# B&R Automation Studio project EFI (part 2)

### IoMap.iom - X20CP1382/IoMap.iom
```iecst
VAR_CONFIG
	Cyclic#4.::X20DIF371_002.DInput[1] AT %IX."X20DIF371_002".DigitalInput01;
	Cyclic#4.::X20DIF371_002.DInput[2] AT %IX."X20DIF371_002".DigitalInput02;
	Cyclic#4.::X20DIF371_002.DInput[3] AT %IX."X20DIF371_002".DigitalInput03;
	Cyclic#4.::X20DIF371_002.DInput[4] AT %IX."X20DIF371_002".DigitalInput04;
	Cyclic#4.::X20DIF371_002.DInput[5] AT %IX."X20DIF371_002".DigitalInput05;
	Cyclic#4.::X20DIF371_002.DInput[6] AT %IX."X20DIF371_002".DigitalInput06;
	Cyclic#4.::X20DIF371_002.DInput[7] AT %IX."X20DIF371_002".DigitalInput07;
	Cyclic#4.::X20DIF371_002.DInput[8] AT %IX."X20DIF371_002".DigitalInput08;
	Cyclic#4.::X20DIF371_002.DInput[9] AT %IX."X20DIF371_002".DigitalInput09;
	Cyclic#4.::X20DIF371_002.DInput[10] AT %IX."X20DIF371_002".DigitalInput10;
	Cyclic#4.::X20DIF371_002.DInput[11] AT %IX."X20DIF371_002".DigitalInput11;
	Cyclic#4.::X20DIF371_002.DInput[12] AT %IX."X20DIF371_002".DigitalInput12;
	Cyclic#4.::X20DIF371_002.DInput[13] AT %IX."X20DIF371_002".DigitalInput13;
	Cyclic#4.::X20DIF371_002.DInput[14] AT %IX."X20DIF371_002".DigitalInput14;
	Cyclic#4.::X20DIF371_002.DInput[15] AT %IX."X20DIF371_002".DigitalInput15;
	Cyclic#4.::X20DIF371_002.DInput[16] AT %IX."X20DIF371_002".DigitalInput16;
	Cyclic#4.::X20DIF371_001.ModuleOk AT %IX."X20DIF371_001".ModuleOk;
	Cyclic#2.::X1.DInput[1] AT %IX."X1".DigitalInput01;
	Cyclic#2.::X1.DInput[2] AT %IX."X1".DigitalInput02;
	Cyclic#2.::X1.DInput[3] AT %IX."X1".DigitalInput03;
	Cyclic#4.::X1.DInput[4] AT %IX."X1".DigitalInput04;
	Cyclic#4.::X1.AInput[1] AT %IW."X1".AnalogInput01;
	Cyclic#4.::X1.AInput[2] AT %IW."X1".AnalogInput02;
	Cyclic#4.::X1.Status01 AT %IB."X1".StatusInput01;
	Cyclic#4.::X2.DInput[1] AT %IX."X2".DigitalInput01;
	Cyclic#4.::X2.DInput[2] AT %IX."X2".DigitalInput02;
	Cyclic#4.::X2.DInput[3] AT %IX."X2".DigitalInput03;
	Cyclic#4.::X2.DInput[4] AT %IX."X2".DigitalInput04;
	Cyclic#4.::X2.DInput[5] AT %IX."X2".DigitalInput05;
	Cyclic#4.::X2.DInput[6] AT %IX."X2".DigitalInput06;
	Cyclic#4.::X2.DInput[7] AT %IX."X2".DigitalInput07;
	Cyclic#4.::X2.DInput[8] AT %IX."X2".DigitalInput08;
	Cyclic#4.::X2.DInput[9] AT %IX."X2".DigitalInput09;
	Cyclic#4.::X2.DInput[10] AT %IX."X2".DigitalInput10;
	Cyclic#4.::X2.DInput[11] AT %IX."X2".DigitalInput11;
	Cyclic#4.::X2.DInput[12] AT %IX."X2".DigitalInput12;
	Cyclic#4.::X2.DInput[13] AT %IX."X2".DigitalInput13;
	Cyclic#4.::X2.DInput[14] AT %IX."X2".DigitalInput14;
	Cyclic#4.::X20DIF371_002.ModuleOk AT %IX."X20DIF371_002".ModuleOk;
	Cyclic#4.::X20DIF371_003.DInput[1] AT %IX."X20DIF371_003".DigitalInput01;
	Cyclic#4.::X20DIF371_003.DInput[2] AT %IX."X20DIF371_003".DigitalInput02;
	Cyclic#4.::X20DIF371_003.DInput[3] AT %IX."X20DIF371_003".DigitalInput03;
	Cyclic#4.::X20DIF371_003.DInput[4] AT %IX."X20DIF371_003".DigitalInput04;
	Cyclic#4.::X20DIF371_003.DInput[5] AT %IX."X20DIF371_003".DigitalInput05;
	Cyclic#4.::X20DIF371_003.DInput[6] AT %IX."X20DIF371_003".DigitalInput06;
	Cyclic#4.::X20DIF371_003.DInput[7] AT %IX."X20DIF371_003".DigitalInput07;
	Cyclic#4.::X20DIF371_003.DInput[8] AT %IX."X20DIF371_003".DigitalInput08;
	Cyclic#4.::X20DIF371_003.DInput[9] AT %IX."X20DIF371_003".DigitalInput09;
	Cyclic#4.::X20DIF371_003.DInput[10] AT %IX."X20DIF371_003".DigitalInput10;
	Cyclic#4.::X20DIF371_003.DInput[11] AT %IX."X20DIF371_003".DigitalInput11;
	Cyclic#4.::X20DIF371_003.DInput[12] AT %IX."X20DIF371_003".DigitalInput12;
	Cyclic#4.::X20DIF371_003.DInput[13] AT %IX."X20DIF371_003".DigitalInput13;
	Cyclic#4.::X20DIF371_003.DInput[14] AT %IX."X20DIF371_003".DigitalInput14;
	Cyclic#4.::X20DIF371_003.DInput[15] AT %IX."X20DIF371_003".DigitalInput15;
	Cyclic#4.::X20DIF371_003.DInput[16] AT %IX."X20DIF371_003".DigitalInput16;
	Cyclic#4.::X20DIF371_004.ModuleOk AT %IX."X20DIF371_004".ModuleOk;
	Cyclic#1.::SiUnitBK1.ModuleOk AT %IX."SI_unit_BK1".ModuleOk;
	Cyclic#1.::SiUnitBK1.NodeStatus AT %IW."SI_unit_BK1".NodeStatus;
	Cyclic#1.::SiUnitBK1.Input01_08 AT %IB."SI_unit_BK1".ReadInout1hTo8h_6000sub1;
	Cyclic#1.::SiUnitBK1.Input09_16 AT %IB."SI_unit_BK1".ReadInput9hTo16h_6000sub2;
	Cyclic#1.::SiUnitBK1.Input17_24 AT %IB."SI_unit_BK1".ReadInput17hTo24h_6000sub3;
	Cyclic#1.::SiUnitBK1.Input25_32 AT %IB."SI_unit_BK1".ReadInput25hTo32h_6000sub4;
	Cyclic#1.::SiUnitBK1.Output01_08 AT %QB."SI_unit_BK1".WriteOutput1hTo8h_6200sub1;
	Cyclic#1.::SiUnitBK1.Output09_16 AT %QB."SI_unit_BK1".WriteOutput9hTo16h_6200sub2;
	Cyclic#1.::SiUnitBK1.Output17_24 AT %QB."SI_unit_BK1".WriteOutput17hTo24h_6200sub3;
	Cyclic#1.::SiUnitBK1.Output25_32 AT %QB."SI_unit_BK1".WriteOutput25hTo32h_6200sub4;
	Cyclic#4.::X3.DInput[5] AT %IX."X3".DigitalInput05;
	Cyclic#4.::X3.DInput[6] AT %IX."X3".DigitalInput06;
	Cyclic#4.::X3.DInput[7] AT %IX."X3".DigitalInput07;
	Cyclic#4.::X3.DOutput[1] AT %QX."X3".DigitalOutput01;
	Cyclic#4.::X3.DOutput[2] AT %QX."X3".DigitalOutput02;
	Cyclic#4.::X3.DOutput[3] AT %QX."X3".DigitalOutput03;
	Cyclic#4.::X3.DOutput[4] AT %QX."X3".DigitalOutput04;
	Cyclic#4.::X3.DOutput[8] AT %QX."X3".DigitalOutput08;
	Cyclic#4.::X3.DOutput[9] AT %QX."X3".DigitalOutput09;
	Cyclic#4.::X3.DOutput[10] AT %QX."X3".DigitalOutput10;
	Cyclic#4.::X3.DOutput[11] AT %QX."X3".DigitalOutput11;
	Cyclic#4.::X3.DOutput[12] AT %QX."X3".DigitalOutput12;
	Cyclic#4.::X20DOF322_005.ModuleOk AT %IX."X20DOF322_005".ModuleOk;
	Cyclic#1.::gIclaNetData[1].xModuleOK AT %IX."ILE1F_BK1".ModuleOk;
	Cyclic#1.::gIclaNetData[1].RPDO4.driveCtrl AT %QB."ILE1F_BK1".Pdo4_driveCtrl_301Esub1;
	Cyclic#1.::gIclaNetData[1].RPDO4.modeCtrl AT %QB."ILE1F_BK1".Pdo4_modeCtrl_301Esub2;
	Cyclic#1.::gIclaNetData[1].TPDO4.modeStat AT %IB."ILE1F_BK1".Pdo4_modeStat_301Esub3;
	Cyclic#1.::gIclaNetData[1].TPDO4.driveStat AT %IW."ILE1F_BK1".Pdo4_driveStat_301Esub4;
	Cyclic#1.::gIclaNetData[1].RPDO4.Ref16 AT %QW."ILE1F_BK1".Pdo4_Ref16_301Esub5;
	Cyclic#1.::gIclaNetData[1].RPDO4.Ref32 AT %QD."ILE1F_BK1".Pdo4_Ref32_301Esub6;
	Cyclic#1.::gIclaNetData[1].TPDO4.Act32 AT %ID."ILE1F_BK1".Pdo4_Act32_301Esub8;
	Cyclic#1.::gIclaNetData[1].TPDO4.Act8 AT %IB."ILE1F_BK1".Pdo4_Act8_301Esub7;
	Cyclic#1.::gAxisStepper[1].DrvIf.iLifeCnt AT %IB."X20SM1436_011".LifeCnt;
	Cyclic#1.::gAxisStepper[1].DrvIf.iDrvOK AT %IX."X20SM1436_011".DrvOk01;
	Cyclic#1.::gAxisStepper[1].DrvIf.oBoostCurrent AT %QX."X20SM1436_011".BoostCurrent01;
	Cyclic#1.::gAxisStepper[1].DrvIf.oStandStillCurrent AT %QX."X20SM1436_011".StandstillCurrent01;
	Cyclic#1.::gAxisStepper[1].DrvIf.oSetTime AT %QW."X20SM1436_011".SetTime01;
	Cyclic#1.::gAxisStepper[1].DiDoIf.iLifeCntDriveEnable AT %IB."X20SM1436_011".LifeCnt;
	Cyclic#1.::gAxisStepper[1].DiDoIf.iLifeCntDriveReady AT %IB."X20SM1436_011".LifeCnt;
	Cyclic#1.::gAxisStepper[1].DiDoIf.iDriveReady AT %IX."X20SM1436_011".DrvOk01;
	Cyclic#1.::gAxisStepper[1].EncIf1.iLifeCnt AT %IB."X20SM1436_011".LifeCnt;
	Cyclic#1.::gAxisStepper[1].EncIf1.iEncOK AT %IX."X20SM1436_011".EncOk01;
	Cyclic#1.::gAxisStepper[1].EncIf1.iActPos AT %IW."X20SM1436_011".ActPos01;
	Cyclic#1.::gAxisStepper[1].EncIf1.iRefPulsePos AT %IW."X20SM1436_011".RefPulsePos01;
	Cyclic#1.::gAxisStepper[1].EncIf1.iRefPulseCnt AT %IB."X20SM1436_011".RefPulseCnt01;
	Cyclic#1.::gAxisStepper[1].EncIf1.iActTime AT %IW."X20SM1436_011".ActTime01;
	Cyclic#1.::X20SM1436_011.ModuleOk AT %IX."X20SM1436_011".ModuleOk;
	Cyclic#1.::gAxisStepper[1].DiDoIf.oDriveEnable AT %QX."X20SM1436_011".DriveEnable01;
	Cyclic#1.::gAxisStepper[1].MotorStep0 AT %QW."X20SM1436_011".Motor1Step0;
	Cyclic#1.::gAxisStepper[2].DrvIf.iLifeCnt AT %IB."X20SM1436_012".LifeCnt;
	Cyclic#1.::gAxisStepper[2].DrvIf.iDrvOK AT %IX."X20SM1436_012".DrvOk01;
	Cyclic#1.::gAxisStepper[2].DrvIf.oBoostCurrent AT %QX."X20SM1436_012".BoostCurrent01;
	Cyclic#1.::gAxisStepper[2].DrvIf.oStandStillCurrent AT %QX."X20SM1436_012".StandstillCurrent01;
	Cyclic#1.::gAxisStepper[2].DrvIf.oSetTime AT %QW."X20SM1436_012".SetTime01;
	Cyclic#1.::gAxisStepper[2].MotorStep0 AT %QW."X20SM1436_012".Motor1Step0;
	Cyclic#1.::gAxisStepper[2].DiDoIf.iLifeCntDriveEnable AT %IB."X20SM1436_012".LifeCnt;
	Cyclic#1.::gAxisStepper[2].DiDoIf.iLifeCntDriveReady AT %IB."X20SM1436_012".LifeCnt;
	Cyclic#1.::gAxisStepper[2].DiDoIf.iDriveReady AT %IX."X20SM1436_012".DrvOk01;
	Cyclic#1.::gAxisStepper[2].DiDoIf.oDriveEnable AT %QX."X20SM1436_012".DriveEnable01;
	Cyclic#1.::gAxisStepper[2].EncIf1.iLifeCnt AT %IB."X20SM1436_012".LifeCnt;
	Cyclic#1.::gAxisStepper[2].EncIf1.iEncOK AT %IX."X20SM1436_012".EncOk01;
	Cyclic#1.::gAxisStepper[2].EncIf1.iActPos AT %IW."X20SM1436_012".ActPos01;
	Cyclic#1.::gAxisStepper[2].EncIf1.iRefPulsePos AT %IW."X20SM1436_012".RefPulsePos01;
	Cyclic#1.::gAxisStepper[2].EncIf1.iRefPulseCnt AT %IB."X20SM1436_012".RefPulseCnt01;
	Cyclic#1.::gAxisStepper[2].EncIf1.iActTime AT %IW."X20SM1436_012".ActTime01;
	Cyclic#1.::X20SM1436_012.ModuleOk AT %IX."X20SM1436_012".ModuleOk;
	Cyclic#4.::X20DIF371_001.DInput[1] AT %IX."X20DIF371_001".DigitalInput01;
	Cyclic#4.::X20DIF371_001.DInput[2] AT %IX."X20DIF371_001".DigitalInput02;
	Cyclic#4.::X20DIF371_001.DInput[3] AT %IX."X20DIF371_001".DigitalInput03;
	Cyclic#4.::X20DIF371_001.DInput[4] AT %IX."X20DIF371_001".DigitalInput04;
	Cyclic#4.::X20DIF371_001.DInput[5] AT %IX."X20DIF371_001".DigitalInput05;
	Cyclic#4.::X20DIF371_001.DInput[6] AT %IX."X20DIF371_001".DigitalInput06;
	Cyclic#4.::X20DIF371_001.DInput[7] AT %IX."X20DIF371_001".DigitalInput07;
	Cyclic#4.::X20DIF371_001.DInput[8] AT %IX."X20DIF371_001".DigitalInput08;
	Cyclic#4.::X20DIF371_001.DInput[9] AT %IX."X20DIF371_001".DigitalInput09;
	Cyclic#4.::X20DIF371_001.DInput[10] AT %IX."X20DIF371_001".DigitalInput10;
	Cyclic#4.::X20DIF371_001.DInput[11] AT %IX."X20DIF371_001".DigitalInput11;
	Cyclic#4.::X20DIF371_001.DInput[12] AT %IX."X20DIF371_001".DigitalInput12;
	Cyclic#4.::X20DIF371_001.DInput[13] AT %IX."X20DIF371_001".DigitalInput13;
	Cyclic#4.::X20DIF371_001.DInput[14] AT %IX."X20DIF371_001".DigitalInput14;
	Cyclic#4.::X20DIF371_001.DInput[15] AT %IX."X20DIF371_001".DigitalInput15;
	Cyclic#4.::X20DIF371_001.DInput[16] AT %IX."X20DIF371_001".DigitalInput16;
	::X20DIF371_003.ModuleOk AT %IX."X20DIF371_003".ModuleOk;
	Cyclic#4.::X20DIF371_004.DInput[1] AT %IX."X20DIF371_004".DigitalInput01;
	Cyclic#4.::X20DIF371_004.DInput[2] AT %IX."X20DIF371_004".DigitalInput02;
	Cyclic#4.::X20DIF371_004.DInput[3] AT %IX."X20DIF371_004".DigitalInput03;
	Cyclic#4.::X20DIF371_004.DInput[4] AT %IX."X20DIF371_004".DigitalInput04;
	Cyclic#4.::X20DIF371_004.DInput[5] AT %IX."X20DIF371_004".DigitalInput05;
	Cyclic#4.::X20DIF371_004.DInput[6] AT %IX."X20DIF371_004".DigitalInput06;
	Cyclic#4.::X20DIF371_004.DInput[7] AT %IX."X20DIF371_004".DigitalInput07;
	Cyclic#4.::X20DIF371_004.DInput[8] AT %IX."X20DIF371_004".DigitalInput08;
	Cyclic#4.::X20DIF371_004.DInput[9] AT %IX."X20DIF371_004".DigitalInput09;
	Cyclic#4.::X20DIF371_004.DInput[10] AT %IX."X20DIF371_004".DigitalInput10;
	Cyclic#4.::X20DIF371_004.DInput[11] AT %IX."X20DIF371_004".DigitalInput11;
	Cyclic#4.::X20DIF371_004.DInput[12] AT %IX."X20DIF371_004".DigitalInput12;
	Cyclic#4.::X20DIF371_004.DInput[13] AT %IX."X20DIF371_004".DigitalInput13;
	Cyclic#4.::X20DIF371_004.DInput[14] AT %IX."X20DIF371_004".DigitalInput14;
	Cyclic#4.::X20DIF371_004.DInput[15] AT %IX."X20DIF371_004".DigitalInput15;
	Cyclic#4.::X20DIF371_004.DInput[16] AT %IX."X20DIF371_004".DigitalInput16;
	Cyclic#4.::X20DOF322_005.DOutput[1] AT %QX."X20DOF322_005".DigitalOutput01;
	Cyclic#4.::X20DOF322_005.DOutput[2] AT %QX."X20DOF322_005".DigitalOutput02;
	Cyclic#4.::X20DOF322_005.DOutput[3] AT %QX."X20DOF322_005".DigitalOutput03;
	Cyclic#4.::X20DOF322_005.DOutput[4] AT %QX."X20DOF322_005".DigitalOutput04;
	Cyclic#4.::X20DOF322_005.DOutput[5] AT %QX."X20DOF322_005".DigitalOutput05;
	Cyclic#4.::X20DOF322_005.DOutput[6] AT %QX."X20DOF322_005".DigitalOutput06;
	Cyclic#4.::X20DOF322_005.DOutput[7] AT %QX."X20DOF322_005".DigitalOutput07;
	Cyclic#4.::X20DOF322_005.DOutput[8] AT %QX."X20DOF322_005".DigitalOutput08;
	Cyclic#4.::X20DOF322_005.DOutput[9] AT %QX."X20DOF322_005".DigitalOutput09;
	Cyclic#4.::X20DOF322_005.DOutput[10] AT %QX."X20DOF322_005".DigitalOutput10;
	Cyclic#4.::X20DOF322_005.DOutput[11] AT %QX."X20DOF322_005".DigitalOutput11;
	Cyclic#4.::X20DOF322_005.DOutput[12] AT %QX."X20DOF322_005".DigitalOutput12;
	Cyclic#4.::X20DOF322_005.DOutput[13] AT %QX."X20DOF322_005".DigitalOutput13;
	Cyclic#4.::X20DOF322_005.DOutput[14] AT %QX."X20DOF322_005".DigitalOutput14;
	Cyclic#4.::X20DOF322_005.DOutput[15] AT %QX."X20DOF322_005".DigitalOutput15;
	Cyclic#4.::X20DOF322_005.DOutput[16] AT %QX."X20DOF322_005".DigitalOutput16;
	::X20DOF322_006.ModuleOk AT %IX."X20DOF322_006".ModuleOk;
	Cyclic#4.::X20DOF322_006.DOutput[1] AT %QX."X20DOF322_006".DigitalOutput01;
	Cyclic#4.::X20DOF322_006.DOutput[2] AT %QX."X20DOF322_006".DigitalOutput02;
	Cyclic#4.::X20DOF322_006.DOutput[3] AT %QX."X20DOF322_006".DigitalOutput03;
	Cyclic#4.::X20DOF322_006.DOutput[4] AT %QX."X20DOF322_006".DigitalOutput04;
	Cyclic#4.::X20DOF322_006.DOutput[5] AT %QX."X20DOF322_006".DigitalOutput05;
	Cyclic#4.::X20DOF322_006.DOutput[6] AT %QX."X20DOF322_006".DigitalOutput06;
	Cyclic#4.::X20DOF322_006.DOutput[7] AT %QX."X20DOF322_006".DigitalOutput07;
	Cyclic#4.::X20DOF322_006.DOutput[8] AT %QX."X20DOF322_006".DigitalOutput08;
	Cyclic#4.::X20DOF322_006.DOutput[9] AT %QX."X20DOF322_006".DigitalOutput09;
	Cyclic#4.::X20DOF322_006.DOutput[10] AT %QX."X20DOF322_006".DigitalOutput10;
	Cyclic#4.::X20DOF322_006.DOutput[11] AT %QX."X20DOF322_006".DigitalOutput11;
	Cyclic#4.::X20DOF322_006.DOutput[12] AT %QX."X20DOF322_006".DigitalOutput12;
	Cyclic#4.::X20DOF322_006.DOutput[13] AT %QX."X20DOF322_006".DigitalOutput13;
	Cyclic#4.::X20DOF322_006.DOutput[14] AT %QX."X20DOF322_006".DigitalOutput14;
	Cyclic#4.::X20DOF322_006.DOutput[15] AT %QX."X20DOF322_006".DigitalOutput15;
	Cyclic#4.::X20DOF322_006.DOutput[16] AT %QX."X20DOF322_006".DigitalOutput16;
	Cyclic#4.::X20AO4622_009.ModuleOk AT %IX."X20AO4622_009".ModuleOk;
	Cyclic#4.::X20AO4622_009.AOutput[1] AT %QW."X20AO4622_009".AnalogOutput01;
	Cyclic#4.::X20AO4622_009.AOutput[2] AT %QW."X20AO4622_009".AnalogOutput02;
	Cyclic#4.::X20AO4622_009.AOutput[3] AT %QW."X20AO4622_009".AnalogOutput03;
	Cyclic#4.::X20AO4622_009.AOutput[4] AT %QW."X20AO4622_009".AnalogOutput04;
	Cyclic#4.::X20AT4222_010.ModuleOk AT %IX."X20AT4222_010".ModuleOk;
	Cyclic#4.::X20AT4222_010.TempInput[1] AT %IW."X20AT4222_010".Temperature01;
	Cyclic#4.::X20AT4222_010.TempInput[2] AT %IW."X20AT4222_010".Temperature02;
	Cyclic#4.::X20AT4222_010.TempInput[3] AT %IW."X20AT4222_010".Temperature03;
	Cyclic#4.::X20AT4222_010.TempInput[4] AT %IW."X20AT4222_010".Temperature04;
	X20AI4322_008.AInput[1] AT %IW."X20AI4322_008".AnalogInput01;
	X20AI4322_008.AInput[2] AT %IW."X20AI4322_008".AnalogInput02;
	X20AI4322_008.AInput[3] AT %IW."X20AI4322_008".AnalogInput03;
	X20AI4322_008.AInput[4] AT %IW."X20AI4322_008".AnalogInput04;
	X20AI4322_008.ModuleOk AT %IX."X20AI4322_008".ModuleOk;
	X20AI4322_008.Status01 AT %IB."X20AI4322_008".StatusInput01;
	::X20AT4222_010.Status01 AT %IB."X20AT4222_010".StatusInput01;
END_VAR
```

### Acp10cfg.ncc - X20CP1382/Motion/Acp10cfg.ncc
```
NcConfiguration (Version=5.15.1, NcSwId=Acp10)
  ACP10CF1_typ:
    cnt_nettrc_rec_drive = 1500
    bufsize_trace_upload = 1200
    tc_nc_man_task = Cyclic #1
    glob_pv_as_ncobject = Yes
    ncsys_dl_broadcast = Yes
    ncsys_dl_acp_reset = Yes
    safemc_log_err_to_ax = Yes
    network_init:
      ncsw_init_execute = Yes
      automatic_execute = Yes
      node_nr_warning = Yes
      net_err_before_ncact = Yes
    nettrc:
      enter_parsecrec = Yes
      enter_ncaction = Yes
      save_ring_startidx = No
    cam_prof_download:
      cam_dat_dl_parallel = No
      tc_cam_dl_parallel = Task class for NC Manager task
    plk_if[0]:
      if_name = IF3
      tc_CycDat_PLCopen = Task class for NC Manager task
      mc_broadcast_extdat = No
    sdc_if[0]:
      if_name = SDC_IF1
      mc_broadcast_size = 800
      mc_broadcast_extdat = No
```

### Acp10map.ncm - X20CP1382/Motion/Acp10map.ncm
```
NcMapping (NcSwId=Acp10, DisabledNodesAreHidden=False)
  NcObject gAxis01 (ModuleId=8V1045.00-2_BELT, Type=ncAXIS, Channel=1, AcoposSimulation=Off, InitParameter=BeltShiel1, AcoposParameter=BeltShield, Disabled=FALSE, ModuleDisabled=FALSE)
  NcObject 8V1045.00-2_ncV_AXIS1 (ModuleId=8V1045.00-2_BELT, Type=ncV_AXIS, Channel=1, Disabled=TRUE, ModuleDisabled=FALSE)
  NcObject gAxis21 (ModuleId=8V1010.50-2_BK1, Type=ncAXIS, Channel=1, AcoposSimulation=Off, InitParameter=BK1_i, AcoposParameter=BK1_a, Disabled=FALSE, ModuleDisabled=FALSE)
  NcObject 8V1016.50-2_ncV_AXIS1 (ModuleId=8V1010.50-2_BK1, Type=ncV_AXIS, Channel=1, Disabled=TRUE, ModuleDisabled=FALSE)
  NcObject gAxisStp01 (ModuleId=X20SM1436_011, ModuleAddress=SDC_IF1.ST1, Type=ncAXIS, Channel=1, AcoposSimulation=Off, InitParameter=SM_i, AcoposParameter=SM_a, AdditionalData=SDC_AX_HwPv="gAxisStepper[1].HW", Disabled=FALSE, ModuleDisabled=FALSE)
  NcObject gAxisStp02 (ModuleId=X20SM1436_012, ModuleAddress=SDC_IF1.ST2, Type=ncAXIS, Channel=1, AcoposSimulation=Off, InitParameter=SM_i, AcoposParameter=SM_a, AdditionalData=SDC_AX_HwPv="gAxisStepper[2].HW", Disabled=FALSE, ModuleDisabled=FALSE)
```

## Configuration 2BK12Bar

CPU X20CP1382, AutomationRuntime B4.83, Build 4.1.2, Safety 1.10, Vc V4.72.6

### Task classes (Cpu.sw)
```
Cyclic#1 (cycle 4000 us, tolerance 0 us):
  InitSteprs <- ExtPack._Motion.StepperCtrl.StepperCtrl_v1.InitStepperX2XCtrl.prg (BuildOptions=-D _IGNORE_CHECKLIB)
  Stepper3L1 <- ExtPack._Motion.StepperCtrl.StepperCtrl_v1.StepperX2XCtrl.prg (BuildOptions=-D _IGNORE_CHECKLIB)
  Stepper3L2 <- ExtPack._Motion.StepperCtrl.StepperCtrl_v1.StepperX2XCtrl.prg (BuildOptions=-D _IGNORE_CHECKLIB)
  Analog <- (binary) (BuildOptions=-D _IGNORE_CHECKLIB)
Cyclic#2 (cycle 12000 us, tolerance 0 us):
  Initialize <- Printer.Config.Initialize.prg (BuildOptions=-D _IGNORE_CHECKLIB)
  InitAxis <- ExtPack._Motion.AxisCtrl.AxisCtrl_v2.InitAxisControl.prg (BuildOptions=-D _IGNORE_CHECKLIB)
  Belt <- ExtPack._Motion.AxisCtrl.AxisCtrl_v2.AxisCtrl.prg (BuildOptions=-D _IGNORE_CHECKLIB)
  BK_A <- ExtPack._Motion.AxisCtrl.AxisCtrl_v2.AxisCtrl.prg (BuildOptions=-D _IGNORE_CHECKLIB)
  BK_B <- ExtPack._Motion.AxisCtrl.AxisCtrl_v2.AxisCtrl.prg (BuildOptions=-D _IGNORE_CHECKLIB)
  Stepper3L <- ExtPack._Motion.AxisCtrl.AxisCtrl_v2.AxisCtrl.prg (BuildOptions=-D _IGNORE_CHECKLIB)
  Gear3L <- ExtPack._Motion.AxisCtrl.AxisCtrl_v2.AxisCtrl.prg (BuildOptions=-D _IGNORE_CHECKLIB)
  InitIcla <- ExtPack._Motion.IclaCtrl.IclaCtrl_v4.InitIclaCtrl.prg (BuildOptions=-D _IGNORE_CHECKLIB)
  IclaBK_A <- ExtPack._Motion.IclaCtrl.IclaCtrl_v4.IclaCtrl.prg (BuildOptions=-D _IGNORE_CHECKLIB)
  IclaBK_B <- ExtPack._Motion.IclaCtrl.IclaCtrl_v4.IclaCtrl.prg (BuildOptions=-D _IGNORE_CHECKLIB)
  Analog_Fas <- ExtPack._Media.AnalogThicknessCtrl.AnalogThicknessCtrl_v1.Analog_Fast.prg (BuildOptions=-D _IGNORE_CHECKLIB)
  nSens_Fast <- ExtPack._Media.nSensorCtrl.nSensorCtrl_v2.nSensorCtrl_Fast.prg (BuildOptions=-D _IGNORE_CHECKLIB)
  Thick_Fast <- ExtPack._Media.ThicknessCtrl.ThicknessCtrl_v2.ThicknessCtrl_Fast.prg (BuildOptions=-D _IGNORE_CHECKLIB)
Cyclic#4 (cycle 32000 us, tolerance 32000 us):
  PhysInp <- Printer.PhysicalMapping.PhysicalMapInputs.prg (BuildOptions=-D _IGNORE_CHECKLIB)
  BlockInp <- Printer.BlockSignalsManager.BlockInputsMapping.prg (BuildOptions=-D _IGNORE_CHECKLIB)  // Physical inputs/outputs block
  ThickPos <- ExtPack._Media.ThicknessCtrl.ThicknessCtrl_v2.ThicknessCtrl.prg (BuildOptions=-D _IGNORE_CHECKLIB)  // Thickness array manager
  Mach_Fast <- Printer.MachineCtrl.MachineCtrl_Fast.prg (BuildOptions=-D _IGNORE_CHECKLIB)
  BeltCtrl <- ExtPack._Transport.BeltCtrl.BeltCtrl_v1.BeltCtrl.prg (BuildOptions=-D _IGNORE_CHECKLIB)  // Belt program
  InitBlockC <- ExtPack.BlockCtrl.BlockCtrl_v1.InitBlockCtrl.prg (BuildOptions=-D _IGNORE_CHECKLIB)  // Init blocks
  Block_BK1 <- ExtPack.BlockCtrl.BlockCtrl_v1.BlockCtrl.prg (BuildOptions=-D _IGNORE_CHECKLIB)
  Block_BK2 <- ExtPack.BlockCtrl.BlockCtrl_v1.BlockCtrl.prg (BuildOptions=-D _IGNORE_CHECKLIB)
  AnalogThic <- ExtPack._Media.AnalogThicknessCtrl.AnalogThicknessCtrl_v1.AnalogThickness.prg (BuildOptions=-D _IGNORE_CHECKLIB)
  nSensorCtr <- ExtPack._Media.nSensorCtrl.nSensorCtrl_v2.nSensorCtrl.prg (BuildOptions=-D _IGNORE_CHECKLIB)
  BlockOut <- Printer.BlockSignalsManager.BlockOutputsMapping.prg (BuildOptions=-D _IGNORE_CHECKLIB)  // Physical HW outputs
  PhysOut <- Printer.PhysicalMapping.PhysicalMapOutputs.prg (BuildOptions=-D _IGNORE_CHECKLIB)
Cyclic#5 (cycle 80000 us, tolerance 80000 us):
  InksInputs <- Printer.InksSignals.InksInputs.prg (BuildOptions=-D _IGNORE_CHECKLIB)  // Physical inputs inks
  InitIndex <- ExtPack.InksCtrl.InksCtrl_v3.InitInksCtrl.prg (BuildOptions=-D _IGNORE_CHECKLIB)
  Inks_01 <- ExtPack.InksCtrl.InksCtrl_v3.InksCtrl.prg (BuildOptions=-D _IGNORE_CHECKLIB)
  Inks_02 <- ExtPack.InksCtrl.InksCtrl_v3.InksCtrl.prg (BuildOptions=-D _IGNORE_CHECKLIB)
  Inks_03 <- ExtPack.InksCtrl.InksCtrl_v3.InksCtrl.prg (BuildOptions=-D _IGNORE_CHECKLIB)
  Inks_04 <- ExtPack.InksCtrl.InksCtrl_v3.InksCtrl.prg (BuildOptions=-D _IGNORE_CHECKLIB)
  Inks_05 <- ExtPack.InksCtrl.InksCtrl_v3.InksCtrl.prg (BuildOptions=-D _IGNORE_CHECKLIB)
  Inks_06 <- ExtPack.InksCtrl.InksCtrl_v3.InksCtrl.prg (BuildOptions=-D _IGNORE_CHECKLIB)
  Inks_07 <- ExtPack.InksCtrl.InksCtrl_v3.InksCtrl.prg (BuildOptions=-D _IGNORE_CHECKLIB)
  Inks_08 <- ExtPack.InksCtrl.InksCtrl_v3.InksCtrl.prg (BuildOptions=-D _IGNORE_CHECKLIB)
  Inks_09 <- ExtPack.InksCtrl.InksCtrl_v3.InksCtrl.prg (BuildOptions=-D _IGNORE_CHECKLIB)
  Inks_10 <- ExtPack.InksCtrl.InksCtrl_v3.InksCtrl.prg (BuildOptions=-D _IGNORE_CHECKLIB)
  Inks_11 <- ExtPack.InksCtrl.InksCtrl_v3.InksCtrl.prg (BuildOptions=-D _IGNORE_CHECKLIB)
  Inks_12 <- ExtPack.InksCtrl.InksCtrl_v3.InksCtrl.prg (BuildOptions=-D _IGNORE_CHECKLIB)
  InksOutput <- Printer.InksSignals.InksOutputs.prg (BuildOptions=-D _IGNORE_CHECKLIB)  // Physical outputs inks
  SafetySamp <- AsSafetySolution.SafetySample.prg (BuildOptions=-D _IGNORE_CHECKLIB)
  EventLogGe <- ExtPack._Tools.EventLog.EventLog_v1.EventLogGen.prg (BuildOptions=-D _IGNORE_CHECKLIB)
  SavePerman <- Printer.Config.SavePermanent.prg (BuildOptions=-D _IGNORE_CHECKLIB)
Cyclic#6 (cycle 88000 us, tolerance 88000 us):
  Mach_Conf <- Printer.Config.MachineConfigurator.prg (BuildOptions=-D _IGNORE_CHECKLIB)  // Printer configurator program
  Mach_Slow <- Printer.MachineCtrl.MachineCtrl_Slow.prg (BuildOptions=-D _IGNORE_CHECKLIB)
Cyclic#7 (cycle 44000 us, tolerance 88000 us):
  PLC2Kernel <- Printer.Comms.PLC2Kernel.prg (BuildOptions=-D _IGNORE_CHECKLIB)  // Comn PLC to kernel
  ServModbus <- ExtPack._Comms.ModbusComms.ModbusComms_v1.ServModbus.prg (BuildOptions=-D _IGNORE_CHECKLIB)
  Kernel2PLC <- Printer.Comms.Kernel2PLC.prg (BuildOptions=-D _IGNORE_CHECKLIB)  // Comns Kernel to PLC
DataObjects: Acp10sys, assl1
NcDataObjects: AcpErrTxt <- AxisTables.AcpErrTxt.dob, acp10etxen <- AxisTables.acp10etxen.dob, BeltA <- AxisTables.BeltP4_a.dob, BeltI <- AxisTables.BeltP4_i.dob, BK1_a <- AxisTables.BK1_a.dob, BK1_i <- AxisTables.BK1_i.dob, SM_a <- AxisTables.SM_a.dob, SM_i <- AxisTables.SM_i.dob
VcDataObjects: Panel1 <- AsSafetySolution.Panel.dob
Binaries: vccnum, vcpdvnc, vccalarm, vccovl, vcshared, vcfile, Panel101, vccstr, vccline, arial, vcpfx20, udbdef, vcchtml, vcgclass, vccbtn, vcrt, vcctext, vcclbox, TCData, Panel102, vccbmp, vcfntttf, vcctrend, vcalarm, vcdsint, vcnet, vccshape, arialbd, vctcal, Panel103, vcmgr, vcdsloc, vcpkat, vccurl, vccdt, vccbar, vcpdsw, vcxml, vcbclass, mvLoader, TCLang, Acp10map, acp10cfg, iomap, User, ashwac, arconfig, Role, ashwd, sysconf, asfw, Visu02, Visu03, Visu01, vccslider, SimVis03, arialxsr, SimVis02, vccgauge, SimVis01, Diagn01, vccpopup, vccddbox, Diagn02, vcchspot, Diagn03, vcpfar00
Libraries: AsCANopen, FBs, Functions, ConvertFun, runtime, brsystem, sys_lib, standard, AsSafety, FileIO, AsXml, astime, asstring, AsFifo, NcGlobal, AsBrStr, MTBasics, MTTypes, MTFilter, AsTCP, AsIecCon, AsIOAcc, AsBrMath, AsEPL, ArEventLog, Acp10_MC, Acp10man, Acp10par, Acp10sim, Acp10sdc, DataObj, EvLogLib, ArProject, BRSE_MB, BRSE_MBT, AxisFunc, AsSem, vcresman, powerlnk, ashw, arssl, AsOpcUas, AsOpcUac, ThickLib
```
